TYPE EventContainer :
STRUCT
	event : FB_Alarm;
	{attribute 'TcEncoding' := 'UTF-8'}
	event_text	: T_MaxString;
END_STRUCT
END_TYPE

(* stored: Version 1.1.0.1, ProductVersion 3.1.4024.15
   DUT EventContainer: Id {b612e6b4-90a5-4f58-b252-1cc5c186438c} *)
